FUNCTION_BLOCK "UNI_TO_GBK"
{ S7_Optimized_Access := 'TRUE' }
VERSION : 0.1
   VAR_INPUT
      UNICODE : Word;
   END_VAR

   VAR_OUTPUT
      GBK : Word;
   END_VAR

   VAR
